INTERFACE I_ITF1

METHOD METH1 : I_ITF1
VAR_INPUT
END_VAR
END_METHOD

PROPERTY Prop1 : I_ITF2
GET
END_GET
END_PROPERTY

END_INTERFACE

(* stored: Version 1.1.0.1, ProductVersion 3.1.4024.12
   Itf I_ITF1: Id {ed93771c-a717-4ce0-aba9-b3f38f5cd6d2}
   Method METH1: Id {b7062bfd-7c35-4ff2-b98b-84d99d3d0db7}
   Property Prop1: Id {eeb3b7b2-05f8-4228-bf38-80030244bdf8}
   Get Get: Id {41b6756a-f53f-47c7-b363-6912d617a094} *)
